TYPE (* logiBUS AI Struct Octal *)
  (* Version 1.0, 2026-05-28, franz *)
  PACKAGE logiBUS::io::AI;
  logiBUS_AI_S_Octal : STRUCT
    Port1 : logiBUS::io::AI::logiBUS_AI_S := (Pin := 255);
    Port2 : logiBUS::io::AI::logiBUS_AI_S := (Pin := 255);
    Port3 : logiBUS::io::AI::logiBUS_AI_S := (Pin := 255);
    Port4 : logiBUS::io::AI::logiBUS_AI_S := (Pin := 255);
    Port5 : logiBUS::io::AI::logiBUS_AI_S := (Pin := 255);
    Port6 : logiBUS::io::AI::logiBUS_AI_S := (Pin := 255);
    Port7 : logiBUS::io::AI::logiBUS_AI_S := (Pin := 255);
    Port8 : logiBUS::io::AI::logiBUS_AI_S := (Pin := 255);
  END_STRUCT;
END_TYPE
